KUKA KRL data list: testglobals.dat

&ACCESS RVO1
&REL 13

DEFDAT  testglobals

GLOBAL ENUM IPO_MODE_T AAA,BBB
GLOBAL STRUC BWDAT REAL VEL1,ACC1,APO_DIST,APO_MODE_T APO_MODE,REAL GEAR_JERK,INT EXAX_IGN
DECL GLOBAL BWDAT BWDEFAULT={VEL 100.000,ACC 100.000,APO_DIST 500.000,APO_MODE #CDIS,GEAR_JERK 100.000,EXAX_IGN 0}
DECL GLOBAL INT ACT_BW_DELAY

ENDDAT
